// Interlock logic for the Dump Chiller
FUNCTION F_ChillerValveEnable : BOOL
VAR_INPUT
END_VAR
VAR_IN_OUT CONSTANT
    stErrors : ST_ErrorStates; // Currently detected errors
END_VAR
VAR
END_VAR

IF stErrors.bHardwareFailure OR stErrors.bLeakDetected THEN
    F_ChillerValveEnable := FALSE;
ELSE
    F_ChillerValveEnable := TRUE;
END_IF

END_FUNCTION

(* stored: Version 1.1.0.1, ProductVersion 3.1.4022.18
   POU F_ChillerValveEnable: Id {eacb95fa-49ef-4c8d-8057-f0d541675cea}, SpecialFunc None *)
